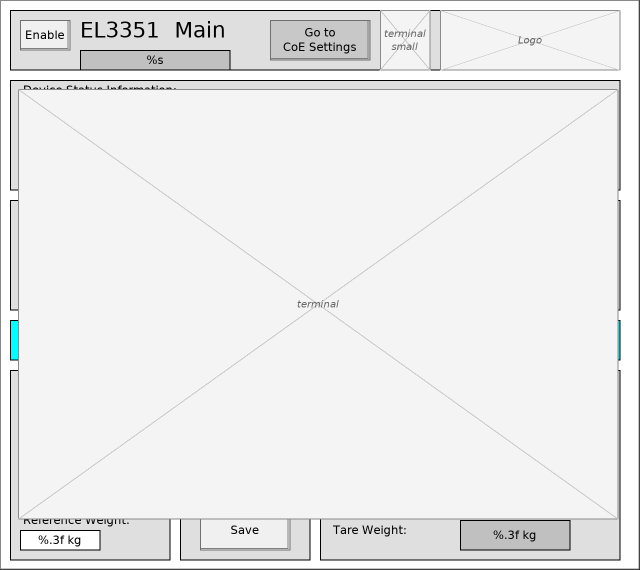
VISUALIZATION VISU_EL3351_BASIC  // 640x570
VAR_IN_OUT
	m_Input_afbEL3351_Index_ : FB_EL3351;
END_VAR
    Rectangle (0,0 640x570)
    Rectangle (10,10 610x60)
    Rectangle (70,10 100x40), "EL3351"
    Image (440,10 180x60), image: Logo
    Image (440,10 180x60), image: Logo
    Rectangle (150,10 100x40), "Main"
    Rectangle (10,370 160x190)
    Rectangle (20,410 100x20), "%.1f kg", text variable: m_Input_afbEL3351_Index_.fbMeasure.rRatedCapacity, input disabled if: (m_Input_afbEL3351_Index_.fbMeasure.nStepCalibrate<>10 AND m_Input_afbEL3351_Index_.fbMeasure.bCalibration) OR NOT m_Input_afbEL3351_Index_.fbMeasure.bUseVisuInputs, colour variable: m_Input_afbEL3351_Index_.fbMeasure.dwColourRatedCapacity
        OnMouseDown: write the text variable via Edit
    Rectangle (20,390 170x20), "Rated Capacity (Emax):"
    Rectangle (20,470 110x20), "Zero Balance:"
    Rectangle (20,490 100x20), "%.4f mV/V", text variable: m_Input_afbEL3351_Index_.fbMeasure.rZeroBalance, input disabled if: (m_Input_afbEL3351_Index_.fbMeasure.bCalibration OR NOT m_Input_afbEL3351_Index_.fbMeasure.bUseVisuInputs) <> 0, colour variable: m_Input_afbEL3351_Index_.fbMeasure.dwColourZeroBalance
        OnMouseDown: write the text variable via Edit
    Rectangle (20,450 100x20), "%.4f mV/V", text variable: m_Input_afbEL3351_Index_.fbMeasure.rRatedOutput, input disabled if: (m_Input_afbEL3351_Index_.fbMeasure.bCalibration OR NOT m_Input_afbEL3351_Index_.fbMeasure.bUseVisuInputs) <> 0, colour variable: m_Input_afbEL3351_Index_.fbMeasure.dwColourRatedOutput
        OnMouseDown: write the text variable via Edit
    Rectangle (20,430 140x20), "Rated Output (Cn):"
    Rectangle (20,370 100x20), "Settings:"
    Button (270,20 100x40), "Go to CoE Settings"
        p3450524324: m_Input_afbEL3351_Index_.dwButtonColour
        tap m_Input_afbEL3351_Index_.bCoEZoom
    Rectangle (10,200 300x110)
    RoundedRectangle (20,250 30x20), "%i", text variable: m_Input_afbEL3351_Index_.fbChannelDiagnosis.bBridgeError, colour variable: m_Input_afbEL3351_Index_.fbChannelDiagnosis.dwBridgeErrorColour
    RoundedRectangle (90,250 30x20), "%i", text variable: m_Input_afbEL3351_Index_.fbChannelDiagnosis.bBridgeUnderrange, colour variable: m_Input_afbEL3351_Index_.fbChannelDiagnosis.dwBridgeUnderrangeColour
    RoundedRectangle (160,250 30x20), "%i", text variable: m_Input_afbEL3351_Index_.fbChannelDiagnosis.bBridgeOverrangerange, colour variable: m_Input_afbEL3351_Index_.fbChannelDiagnosis.dwBridgeOverrangerangeColour
    Rectangle (20,230 50x20), "Error:"
    Rectangle (70,200 190x30), "Bridge Status (Channel 1):"
    Rectangle (320,200 300x110)
    RoundedRectangle (230,250 30x20), "%i", text variable: m_Input_afbEL3351_Index_.fbChannelDiagnosis.bBridgeState, colour variable: m_Input_afbEL3351_Index_.fbChannelDiagnosis.dwBridgeStateColour
    Rectangle (220,230 110x20), "TxPDO State:"
    Rectangle (150,230 90x20), "Overrange:"
    Rectangle (70,230 100x20), "Underrange:"
    Rectangle (380,200 180x30), "Supply Status (Channel 2):"
    RoundedRectangle (330,250 30x20), "%i", text variable: m_Input_afbEL3351_Index_.fbChannelDiagnosis.bSupplyError, colour variable: m_Input_afbEL3351_Index_.fbChannelDiagnosis.dwSupplyErrorColour
    RoundedRectangle (400,250 30x20), "%i", text variable: m_Input_afbEL3351_Index_.fbChannelDiagnosis.bSupplyUnderrange, colour variable: m_Input_afbEL3351_Index_.fbChannelDiagnosis.dwSupplyUnderrangeColour
    RoundedRectangle (470,250 30x20), "%i", text variable: m_Input_afbEL3351_Index_.fbChannelDiagnosis.bSupplyOverrangerange, colour variable: m_Input_afbEL3351_Index_.fbChannelDiagnosis.dwSupplyOverrangerangeColour
    RoundedRectangle (540,250 30x20), "%i", text variable: m_Input_afbEL3351_Index_.fbChannelDiagnosis.bSupplyState, colour variable: m_Input_afbEL3351_Index_.fbChannelDiagnosis.dwSupplyStateColour
    Rectangle (330,230 50x20), "Error:"
    Rectangle (380,230 100x20), "Underrange:"
    Rectangle (460,230 90x20), "Overrange:"
    Rectangle (530,230 110x20), "TxPDO State:"
    Rectangle (330,280 120x20), "Supply Voltage:"
    Rectangle (470,280 110x20), "%.3f V", text variable: m_Input_afbEL3351_Index_.fbMeasure.rUref
    Rectangle (20,280 120x20), "Bridge Voltage:"
    Rectangle (150,280 110x20), "%.3f mV", text variable: m_Input_afbEL3351_Index_.fbMeasure.rUdiff
    Rectangle (10,320 610x40), "%s", text variable: m_Input_afbEL3351_Index_.fbMeasure.sSettings, colour variable: P_LoadCell.fbColours.dwColour
    Rectangle (180,370 130x190)
    Rectangle (20,530 80x20), "%.3f kg", text variable: m_Input_afbEL3351_Index_.fbMeasure.rReferenceWeight, input disabled if: m_Input_afbEL3351_Index_.fbMeasure.nStepCalibrate<>30 OR NOT m_Input_afbEL3351_Index_.fbMeasure.bCalibration, colour variable: m_Input_afbEL3351_Index_.fbMeasure.dwColourReferenceWeight
        OnMouseDown: write the text variable via Edit
    Rectangle (20,510 130x20), "Reference Weight:"
    Button (200,510 90x40), "Save", input disabled if: NOT m_Input_afbEL3351_Index_.fbMeasure.bCalibration
        p3450524324: m_Input_afbEL3351_Index_.fbMeasure.dwColourSave
        tap m_Input_afbEL3351_Index_.fbMeasure.bNextStep
    Button (200,460 90x40), "Start Calibration", input disabled if: NOT m_Input_afbEL3351_Index_.fbMeasure.bCalibration
        p3450524324: m_Input_afbEL3351_Index_.fbMeasure.dwColourStartCalibration
        tap m_Input_afbEL3351_Index_.fbMeasure.bStartCalibration
    Button (200,410 90x40), "Calibration Mode", pressed state: m_Input_afbEL3351_Index_.fbMeasure.bCalibration
        p3450524324: m_Input_afbEL3351_Index_.dwButtonColour
        toggle m_Input_afbEL3351_Index_.fbMeasure.bCalibration
    Rectangle (190,370 100x20), "Calibration:"
    Rectangle (320,370 300x190)
    Rectangle (460,390 110x30), "%.3f kg", text variable: m_Input_afbEL3351_Index_.fbMeasure.rGrossWeight, colour variable: m_Input_afbEL3351_Index_.fbMeasure.dwColourWeight
    Rectangle (330,370 160x20), "Measuring Function:"
    Rectangle (330,400 140x20), "Gross Weight:"
    Button (330,430 90x40), "Set Tare weight"
        p3450524324: m_Input_afbEL3351_Index_.dwButtonColour
        tap m_Input_afbEL3351_Index_.fbMeasure.bSetTare
    Rectangle (460,480 110x30), "%.3f kg", text variable: m_Input_afbEL3351_Index_.fbMeasure.rNetWeight, colour variable: m_Input_afbEL3351_Index_.fbMeasure.dwTareColour
    Rectangle (330,480 100x20), "Net Weight:"
    Button (430,430 90x40), "Reset Tare weight"
        p3450524324: m_Input_afbEL3351_Index_.dwButtonColour
        tap m_Input_afbEL3351_Index_.fbMeasure.bResetTare
    Rectangle (330,520 100x20), "Tare Weight:"
    Rectangle (460,520 110x30), "%.3f kg", text variable: m_Input_afbEL3351_Index_.fbMeasure.rTareWeight, colour variable: m_Input_afbEL3351_Index_.fbMeasure.dwTareColour
    Button (20,20 50x30), "Enable", pressed state: m_Input_afbEL3351_Index_.bEnable
        p3450524324: m_Input_afbEL3351_Index_.dwButtonColour
        toggle m_Input_afbEL3351_Index_.bEnable
    Image (380,10 50x60), image: terminalsmall
        toggle m_Input_afbEL3351_Index_.bConnection
    Rectangle (10,80 610x110)
    Rectangle (20,80 190x20), "Device Status Information:"
    Rectangle (230,120 300x20), "%s", text variable: m_Input_afbEL3351_Index_.fbTerminalDiagnosis.sState, colour variable: m_Input_afbEL3351_Index_.fbTerminalDiagnosis.dwStateStatusColour
    Rectangle (20,120 150x20), "%s", text variable: m_Input_afbEL3351_Index_.fbTerminalDiagnosis.sWorkingState, colour variable: m_Input_afbEL3351_Index_.fbTerminalDiagnosis.dwWcStateColour
    Rectangle (20,160 580x20), "%s", text variable: m_Input_afbEL3351_Index_.fbTerminalDiagnosis.sStateStatusAll, colour variable: m_Input_afbEL3351_Index_.fbTerminalDiagnosis.dwStateStatusAllColour
    Rectangle (20,100 90x20), "WcState:"
    Rectangle (230,100 120x20), "InfoData State:"
    Rectangle (20,140 70x20), "Errors:"
    Rectangle (80,50 150x20), "%s", text variable: m_Input_afbEL3351_Index_.sShowTerminalNumber
    Image (18,89 600x430), invisible if: NOT m_Input_afbEL3351_Index_.bConnection, image: terminal
END_VISUALIZATION

(* stored: Version 1.1.0.1, ProductVersion 3.1.4024.12
   Visu VISU_EL3351_BASIC: Id {3f7f07f5-ddc4-466c-9e93-00e5c3b66354} *)
